FUNCTION_BLOCK CylinderVSens (* Composite Function Block Type *)
  (* Standard: 61499-2 *)
  (* Version 0.0, 5/28/2016, Andrei, nxtControl GmbH, template *)
  PACKAGE Main;
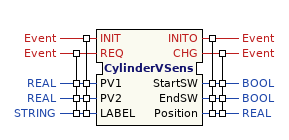
  EVENT_INPUT
    INIT WITH PV1, PV2, LABEL;
    REQ WITH PV1, PV2, LABEL; (* Normal Execution Request *)
  END_EVENT
  EVENT_OUTPUT
    INITO WITH StartSW, EndSW, Position;
    CHG WITH StartSW, EndSW, Position; (* Execution Confirmation *)
  END_EVENT
  VAR_INPUT
    PV1 : REAL; (* Input event qualifier *)
    PV2 : REAL;
    LABEL : STRING;
  END_VAR
  VAR_OUTPUT
    StartSW : BOOL; (* Output event qualifier *)
    EndSW : BOOL;
    Position : REAL;
  END_VAR
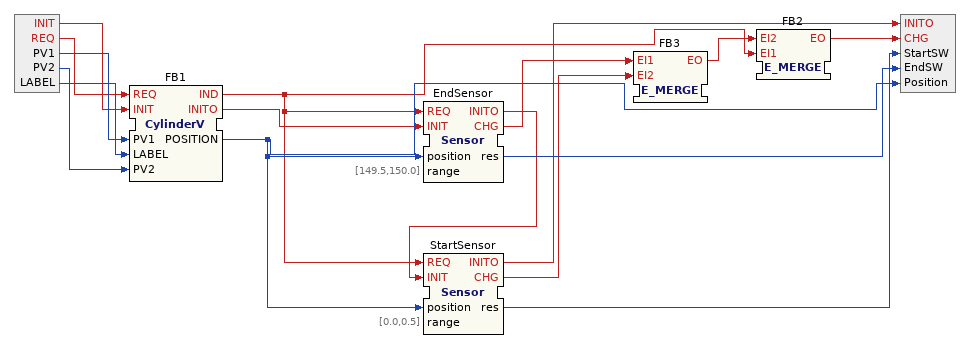
  FBS
    EndSensor : Sensor(range := [149.5,150.0]);
    StartSensor : Sensor(range := [0.0,0.5]);
    FB1 : CylinderV;
    FB2 : E_MERGE;
    FB3 : E_MERGE;
  END_FBS
  EVENT_CONNECTIONS
    REQ TO FB1.REQ;
    FB1.IND TO EndSensor.REQ;
    FB1.IND TO StartSensor.REQ;
    FB2.EO TO CHG;
    INIT TO FB1.INIT;
    StartSensor.INITO TO INITO;
    FB1.INITO TO EndSensor.INIT;
    EndSensor.INITO TO StartSensor.INIT;
    EndSensor.CHG TO FB3.EI1;
    StartSensor.CHG TO FB3.EI2;
    FB3.EO TO FB2.EI2;
    FB1.IND TO FB2.EI1;
  END_CONNECTIONS
  DATA_CONNECTIONS
    PV1 TO FB1.PV1;
    LABEL TO FB1.LABEL;
    PV2 TO FB1.PV2;
    FB1.POSITION TO EndSensor.position;
    StartSensor.res TO StartSW;
    FB1.POSITION TO StartSensor.position;
    FB1.POSITION TO Position;
    EndSensor.res TO EndSW;
  END_CONNECTIONS
END_FUNCTION_BLOCK
